FUNCTION_BLOCK FB_ScaleDevice
VAR_INPUT
    sRemoteHost 	: STRING := '192.168.1.100';
    nRemotePort 	: UINT 	 := 8001;
	bExecuteRequest : BOOL;
	rLastWeight     : LREAL;
END_VAR

VAR_OUTPUT
	bWeightReady : BOOL;
    bBusy        : BOOL;
    bError       : BOOL;
    nErrorID     : UDINT;
END_VAR

VAR
    fbTcpClient     : FB_TcpClient;
   
    bRequestDone    : BOOL;
    sRawResponse    : STRING(255);
    
    sLastMessage    : STRING(255);
END_VAR

// Continous call to keep the function block ready for communication 
IF bExecuteRequest OR fbTcpClient.bBusy THEN
	fbTcpClient(
		sRemoteHost := sRemoteHost,
		nRemotePort := nRemotePort,
		bExecute := bExecuteRequest,
		tStateDelay := T#500MS,
		bConnectionDone => bRequestDone,
		sResponse => sRawResponse,
		bError => bError,
		nErrorID => nErrorID
	);
END_IF

// Done and Reset flags
IF fbTcpClient.bConnectionDone THEN
    bExecuteRequest := FALSE;
    rLastWeight := F_ParseWeight(sRawResponse);
    sLastMessage := CONCAT('Weight: ', LREAL_TO_STRING(rLastWeight));
	bWeightReady := TRUE;
END_IF

METHOD RequestWeight : LREAL
VAR_OUTPUT
    bSuccess : BOOL;
    sMessage : STRING;
END_VAR
// Triggering fbTcpClient
IF NOT bExecuteRequest AND NOT fbTcpClient.bBusy THEN
    bExecuteRequest := TRUE;
END_IF
// Releasing fbTcpClient 
IF fbTcpClient.bConnectionDone THEN
    RequestWeight := rLastWeight;
    bSuccess := TRUE;
    sMessage := sLastMessage;
ELSE
    bSuccess := FALSE;
END_IF
END_METHOD

METHOD Reset : BOOL
VAR_INPUT
END_VAR
bWeightReady := FALSE;
bBusy        := FALSE;
bError       := FALSE;
nErrorID     := 0;
bExecuteRequest := FALSE;
bRequestDone    := FALSE;
sRawResponse    := '';
rLastWeight     := 0.0;
sLastMessage    := '';

IF fbTcpClient.Reset() AND NOT bWeightReady THEN
	Reset := TRUE;
ELSE
	Reset := FALSE;
END_IF
END_METHOD

END_FUNCTION_BLOCK

(* stored: Version 1.1.0.1, ProductVersion 3.1.4024.15
   POU FB_ScaleDevice: Id {61aa2783-8d7b-4a50-a982-014b2d41abdc}, SpecialFunc None
   Method RequestWeight: Id {cd501a59-3fb3-4ee3-b78a-6533885392ec}
   Method Reset: Id {5ccb7417-dde1-4fb5-b36f-0de8a7f97a72} *)
